// TIA Portal V19 export
DATA_BLOCK "MeasuredValues"   // DB110
{ S7_Optimized_Access := 'TRUE' }
AUTHOR : OPA_8160
FAMILY : ANALOG
NAME : ANA_INPU
VERSION : 0.0
// stored: AutoNumber false, MemoryReserve 0
   VAR RETAIN
      TT0176REAL : Real := 124.8148;   // TT 01.76
      TT0178REAL : Real := 127.5;   // TT 01.78
      TT0160REAL : Real := 63.05556;   // TT 01.60
      TT0172REAL : Real := 26.66667;   // TT 01.72
      TT0163REAL : Real := 130.0;   // TT 01.63
      PT0167REAL : Real := 2.480903;   // PT 01.67
      WT0169REAL : Real := 99.82639;   // WT 01.69
      TT0180REAL : Real := 21.94444;   // TT 01.80
      CT0182REAL : Real := -0.1446759;   // CT 01.82
      TT0950REAL : Real := 0.0;   // TT 09.50
      TT0951REAL : Real := 0.0;   // TT 09.51
   END_VAR
BEGIN
END_DATA_BLOCK
